{attribute 'GeneratedUsingTerminal: EK1100-0000-0018'}
{attribute addProperty BoxType "EK1100-0000-0018"}
{attribute addProperty Id "Beckhoff_ELXxxxxEK1122Beckhoff_ELXxxxxEK1122_D1E25D712A_0001_ELX1052_0000_0016ELX1052_FE4CEFB88A_0002_ELX1054_0000_0016ELX1054_91588CA916A_0003_ELX1058_0000_0016ELX1058_64CB4C7B28A_0004_ELX2002_0000_0016ELX2002_22AF7D925A_0005_ELX2008_0000_0016ELX2008_D86968E311A_0006_ELX3152_0000_0016ELX3152_CC62AFB732A_0007_ELX3152_0000_0017ELX3152_CC62AFB732A_0008_ELX3152_0090_0016ELX3152_CC62AFB732A_0009_ELX3152_0090_0017ELX3152_CC62AFB732A_0010_ELX3158_0000_0016ELX3158_5798389192A_0011_ELX3181_0000_0016ELX3181_59E7F0B828A_0012_ELX3181_0000_0017ELX3181_59E7F0B828A_0013_ELX3202_0000_0016ELX3202_14BDD8A530A_0014_ELX3202_0090_0016ELX3202_14BDD8A530A_0015_ELX3204_0000_0016ELX3204_6DF7478348A_0016_ELX3204_0090_0016ELX3204_6DF7478348A_0017_ELX3252_0000_0016ELX3252_7E6368AC26A_0018_ELX3312_0000_0016ELX3312_1587323830A_0019_ELX3312_0090_0016ELX3312_1587323830A_0020_ELX3314_0000_0016ELX3314_6BF23D5548A_0021_ELX3314_0090_0016ELX3314_6BF23D5548A_0022_ELX3351_0000_0016ELX3351_7F234E6326A_0023_ELX3351_0090_0016ELX3351_7F234E6326A_0024_ELX4154_0000_0016ELX4154_F6F08E1219A_0025_ELX4181_0000_0016ELX4181_CF98482419A_0026_ELX4181_0000_0017ELX4181_CF98482419A_0027_ELX5151_0000_0016ELX5151_5B556A9025A_0028_ELX5151_0090_0016ELX5151_5B556A9025A_0030_ELX9410_0000_0016ELX9410_0DA715C26A_0031_ELX9410_0000_0017ELX9410_0DA715C26A_0032_ELX9410_0000_0018ELX9410_D987D9F46A_0033_ELX9560_0000_0016ELX9560_BA4910676A_0034_ELX9560_0000_0017ELX9560_BA4910676A_0035_ELX9560_0000_0018ELX9560_C05BDD366"}
{attribute addProperty CRC "3115172767"}
{attribute addProperty Size "879"}
TYPE Beckhoff_ELXxxxx_B9ADC39F EXTENDS EK1100_AB5A9467 :
STRUCT
	{attribute addProperty Name "Beckhoff_ELXxxxxEK1122"}
	{attribute addProperty PreviousPort "Beckhoff ELXxxxx : B"}
	Beckhoff_ELXxxxxEK1122 : Beckhoff_ELXxxxxEK1122_D1E25D71;
	{attribute addProperty Name "A_0001_ELX1052_0000_0016"}
	{attribute addProperty PreviousPort "Beckhoff ELXxxxxEK1122 : C"}
	A_0001_ELX1052_0000_0016 : ELX1052_FE4CEFB8;
	{attribute addProperty Name "A_0002_ELX1054_0000_0016"}
	{attribute addProperty PreviousPort "A_0001(ELX1052-0000-0016) : B"}
	A_0002_ELX1054_0000_0016 : ELX1054_91588CA9;
	{attribute addProperty Name "A_0003_ELX1058_0000_0016"}
	{attribute addProperty PreviousPort "A_0002(ELX1054-0000-0016) : B"}
	A_0003_ELX1058_0000_0016 : ELX1058_64CB4C7B;
	{attribute addProperty Name "A_0004_ELX2002_0000_0016"}
	{attribute addProperty PreviousPort "A_0003(ELX1058-0000-0016) : B"}
	A_0004_ELX2002_0000_0016 : ELX2002_22AF7D92;
	{attribute addProperty Name "A_0005_ELX2008_0000_0016"}
	{attribute addProperty PreviousPort "A_0004(ELX2002-0000-0016) : B"}
	A_0005_ELX2008_0000_0016 : ELX2008_D86968E3;
	{attribute addProperty Name "A_0006_ELX3152_0000_0016"}
	{attribute addProperty PreviousPort "A_0005(ELX2008-0000-0016) : B"}
	A_0006_ELX3152_0000_0016 : ELX3152_CC62AFB7;
	{attribute addProperty Name "A_0007_ELX3152_0000_0017"}
	{attribute addProperty PreviousPort "A_0006(ELX3152-0000-0016) : B"}
	A_0007_ELX3152_0000_0017 : ELX3152_CC62AFB7;
	{attribute addProperty Name "A_0008_ELX3152_0090_0016"}
	{attribute addProperty PreviousPort "A_0007(ELX3152-0000-0017) : B"}
	A_0008_ELX3152_0090_0016 : ELX3152_CC62AFB7;
	{attribute addProperty Name "A_0009_ELX3152_0090_0017"}
	{attribute addProperty PreviousPort "A_0008(ELX3152-0090-0016) : B"}
	A_0009_ELX3152_0090_0017 : ELX3152_CC62AFB7;
	{attribute addProperty Name "A_0010_ELX3158_0000_0016"}
	{attribute addProperty PreviousPort "A_0009(ELX3152-0090-0017) : B"}
	A_0010_ELX3158_0000_0016 : ELX3158_57983891;
	{attribute addProperty Name "A_0011_ELX3181_0000_0016"}
	{attribute addProperty PreviousPort "A_0010(ELX3158-0000-0016) : B"}
	A_0011_ELX3181_0000_0016 : ELX3181_59E7F0B8;
	{attribute addProperty Name "A_0012_ELX3181_0000_0017"}
	{attribute addProperty PreviousPort "A_0011(ELX3181-0000-0016) : B"}
	A_0012_ELX3181_0000_0017 : ELX3181_59E7F0B8;
	{attribute addProperty Name "A_0013_ELX3202_0000_0016"}
	{attribute addProperty PreviousPort "A_0012(ELX3181-0000-0017) : B"}
	A_0013_ELX3202_0000_0016 : ELX3202_14BDD8A5;
	{attribute addProperty Name "A_0014_ELX3202_0090_0016"}
	{attribute addProperty PreviousPort "A_0013(ELX3202-0000-0016) : B"}
	A_0014_ELX3202_0090_0016 : ELX3202_14BDD8A5;
	{attribute addProperty Name "A_0015_ELX3204_0000_0016"}
	{attribute addProperty PreviousPort "A_0014(ELX3202-0090-0016) : B"}
	A_0015_ELX3204_0000_0016 : ELX3204_6DF74783;
	{attribute addProperty Name "A_0016_ELX3204_0090_0016"}
	{attribute addProperty PreviousPort "A_0015(ELX3204-0000-0016) : B"}
	A_0016_ELX3204_0090_0016 : ELX3204_6DF74783;
	{attribute addProperty Name "A_0017_ELX3252_0000_0016"}
	{attribute addProperty PreviousPort "A_0016(ELX3204-0090-0016) : B"}
	A_0017_ELX3252_0000_0016 : ELX3252_7E6368AC;
	{attribute addProperty Name "A_0018_ELX3312_0000_0016"}
	{attribute addProperty PreviousPort "A_0017(ELX3252-0000-0016) : B"}
	A_0018_ELX3312_0000_0016 : ELX3312_15873238;
	{attribute addProperty Name "A_0019_ELX3312_0090_0016"}
	{attribute addProperty PreviousPort "A_0018(ELX3312-0000-0016) : B"}
	A_0019_ELX3312_0090_0016 : ELX3312_15873238;
	{attribute addProperty Name "A_0020_ELX3314_0000_0016"}
	{attribute addProperty PreviousPort "A_0019(ELX3312-0090-0016) : B"}
	A_0020_ELX3314_0000_0016 : ELX3314_6BF23D55;
	{attribute addProperty Name "A_0021_ELX3314_0090_0016"}
	{attribute addProperty PreviousPort "A_0020(ELX3314-0000-0016) : B"}
	A_0021_ELX3314_0090_0016 : ELX3314_6BF23D55;
	{attribute addProperty Name "A_0022_ELX3351_0000_0016"}
	{attribute addProperty PreviousPort "A_0021(ELX3314-0090-0016) : B"}
	A_0022_ELX3351_0000_0016 : ELX3351_7F234E63;
	{attribute addProperty Name "A_0023_ELX3351_0090_0016"}
	{attribute addProperty PreviousPort "A_0022(ELX3351-0000-0016) : B"}
	A_0023_ELX3351_0090_0016 : ELX3351_7F234E63;
	{attribute addProperty Name "A_0024_ELX4154_0000_0016"}
	{attribute addProperty PreviousPort "A_0023(ELX3351-0090-0016) : B"}
	A_0024_ELX4154_0000_0016 : ELX4154_F6F08E12;
	{attribute addProperty Name "A_0025_ELX4181_0000_0016"}
	{attribute addProperty PreviousPort "A_0024(ELX4154-0000-0016) : B"}
	A_0025_ELX4181_0000_0016 : ELX4181_CF984824;
	{attribute addProperty Name "A_0026_ELX4181_0000_0017"}
	{attribute addProperty PreviousPort "A_0025(ELX4181-0000-0016) : B"}
	A_0026_ELX4181_0000_0017 : ELX4181_CF984824;
	{attribute addProperty Name "A_0027_ELX5151_0000_0016"}
	{attribute addProperty PreviousPort "A_0026(ELX4181-0000-0017) : B"}
	A_0027_ELX5151_0000_0016 : ELX5151_5B556A90;
	{attribute addProperty Name "A_0028_ELX5151_0090_0016"}
	{attribute addProperty PreviousPort "A_0027(ELX5151-0000-0016) : B"}
	A_0028_ELX5151_0090_0016 : ELX5151_5B556A90;
	{attribute addProperty Name "A_0030_ELX9410_0000_0016"}
	{attribute addProperty PreviousPort "A_0028(ELX5151-0090-0016) : B"}
	A_0030_ELX9410_0000_0016 : ELX9410_0DA715C2;
	{attribute addProperty Name "A_0031_ELX9410_0000_0017"}
	{attribute addProperty PreviousPort "A_0030(ELX9410-0000-0016) : B"}
	A_0031_ELX9410_0000_0017 : ELX9410_0DA715C2;
	{attribute addProperty Name "A_0032_ELX9410_0000_0018"}
	{attribute addProperty PreviousPort "A_0031(ELX9410-0000-0017) : B"}
	A_0032_ELX9410_0000_0018 : ELX9410_D987D9F4;
	{attribute addProperty Name "A_0033_ELX9560_0000_0016"}
	{attribute addProperty PreviousPort "A_0032(ELX9410-0000-0018) : B"}
	A_0033_ELX9560_0000_0016 : ELX9560_BA491067;
	{attribute addProperty Name "A_0034_ELX9560_0000_0017"}
	{attribute addProperty PreviousPort "A_0033(ELX9560-0000-0016) : B"}
	A_0034_ELX9560_0000_0017 : ELX9560_BA491067;
	{attribute addProperty Name "A_0035_ELX9560_0000_0018"}
	{attribute addProperty PreviousPort "A_0034(ELX9560-0000-0017) : B"}
	A_0035_ELX9560_0000_0018 : ELX9560_C05BDD36;
END_STRUCT
END_TYPE

(* stored: Version 1.2.0.0, ProductVersion 3.1.4024.9
   DUT Beckhoff_ELXxxxx_B9ADC39F: Id {02594ee5-f7c8-4522-a185-d9bcfaf6c722} *)
